FUNCTION_BLOCK KeepCurrOpCdt (* Basic Function Block Type *)
  (* Standard: 61499-2 *)
  (* Version 0.0, 8/20/2024, SESA713705, Schneider Electric, Template *)
  PACKAGE SE.Nereda;
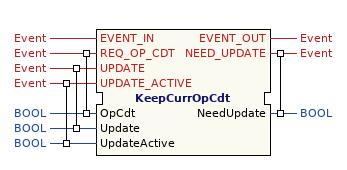
  EVENT_INPUT
    EVENT_IN;
    REQ_OP_CDT WITH OpCdt;
    UPDATE WITH Update;
    UPDATE_ACTIVE WITH UpdateActive;
  END_EVENT
  EVENT_OUTPUT
    EVENT_OUT;
    NEED_UPDATE WITH NeedUpdate;
  END_EVENT
  VAR_INPUT
    OpCdt : BOOL;
    Update : BOOL;
    UpdateActive : BOOL;
  END_VAR
  VAR_OUTPUT
    NeedUpdate : BOOL;
  END_VAR
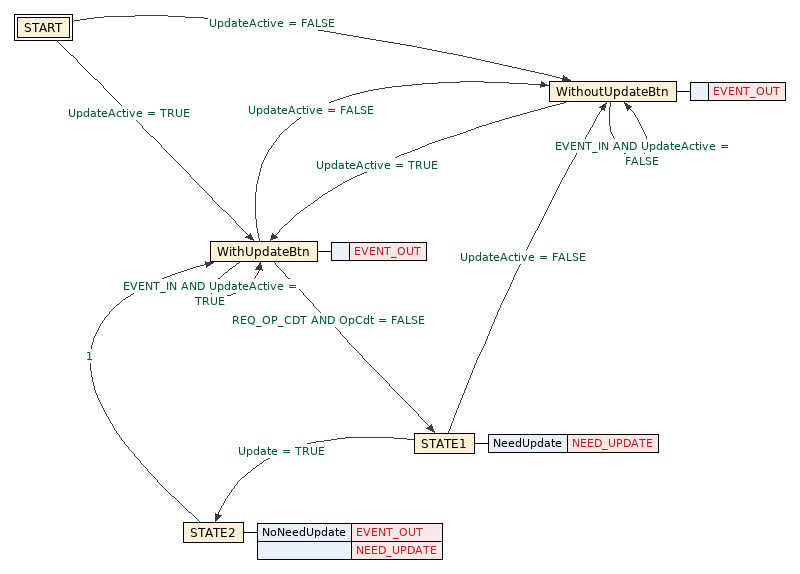
  EC_STATES
    START; (* Initial State *)
    WithUpdateBtn : -> EVENT_OUT;
    STATE1 : NeedUpdate -> NEED_UPDATE;
    STATE2 : NoNeedUpdate -> EVENT_OUT, -> NEED_UPDATE;
    WithoutUpdateBtn : -> EVENT_OUT;
  END_STATES
  EC_TRANSITIONS
    START TO WithUpdateBtn := UpdateActive = TRUE;
    WithUpdateBtn TO STATE1 := REQ_OP_CDT AND OpCdt = FALSE;
    WithUpdateBtn TO WithUpdateBtn := EVENT_IN AND UpdateActive = TRUE;
    STATE1 TO STATE2 := Update = TRUE;
    STATE2 TO WithUpdateBtn := 1;
    START TO WithoutUpdateBtn := UpdateActive = FALSE;
    WithUpdateBtn TO WithoutUpdateBtn := UpdateActive = FALSE;
    STATE1 TO WithoutUpdateBtn := UpdateActive = FALSE;
    WithoutUpdateBtn TO WithUpdateBtn := UpdateActive = TRUE;
    WithoutUpdateBtn TO WithoutUpdateBtn := EVENT_IN AND UpdateActive = FALSE;
  END_TRANSITIONS
  ALGORITHM NeedUpdate IN ST:
;
NeedUpdate := TRUE;
  END_ALGORITHM
  ALGORITHM NoNeedUpdate IN ST:
;
NeedUpdate := FALSE;
  END_ALGORITHM
END_FUNCTION_BLOCK
